FUNCTION_BLOCK CmdVentAeration_HMI (* Service Interface Function Block Type *)
  (* Standard: 61499-2 *)
  (* Version 0.0, 6/7/2026, Schneider Electric, template *)
  PACKAGE SE.Nereda;
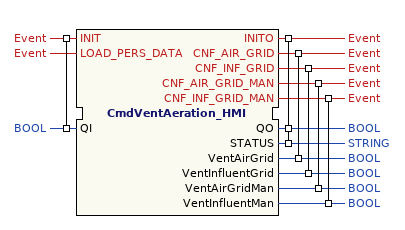
  EVENT_INPUT
    INIT WITH QI;
    LOAD_PERS_DATA;
  END_EVENT
  EVENT_OUTPUT
    INITO WITH QO, STATUS;
    CNF_AIR_GRID WITH VentAirGrid;
    CNF_INF_GRID WITH VentInfluentGrid;
    CNF_AIR_GRID_MAN WITH VentAirGridMan;
    CNF_INF_GRID_MAN WITH VentInfluentMan;
  END_EVENT
  VAR_INPUT
    QI : BOOL;
  END_VAR
  VAR_OUTPUT
    QO : BOOL; (* Event Output Qualifier *)
    STATUS : STRING; (* Service Status *)
    VentAirGrid : BOOL;
    VentInfluentGrid : BOOL;
    VentAirGridMan : BOOL;
    VentInfluentMan : BOOL;
  END_VAR
  SERVICE /
    SEQUENCE 
    END_SEQUENCE
  END_SERVICE
END_FUNCTION_BLOCK
